TYPE Vec7i : ARRAY[1..7] OF INT; END_TYPE

(* stored: Version 1.1.0.1, ProductVersion 3.1.4024.12
   DUT Vec7i: Id {25529931-fd19-4f2c-bc31-0c98dfd28ab0} *)
